(* Logix 5000 project; controller Universal_Device_Info_AOI_V0_1 vendor 1 type 14 code 176 rev 32.11; software revision 32.00; part 2 of 3 *)
(* tags used below, declared in another part *)
   Port : INT;
   Common_Data : Turck_IOLink_Common_Data;
   Universal_IOLink_Info : Universal_IOLink_Info;
   StartupDone : BOOL;
   Done : DINT;
   Error : DINT;
   Active : DINT;
   Pending : DINT;
   Pending_or_Active : DINT;
   MyTicketNum : DINT[32];
   Read_ONS : DINT;
   ReadRequest : DINT;
   Read : DINT;
   DoneCount : DINT;
   Status : DINT;
   ErrorCount : DINT;
   Update_Data : BOOL;
(* Universal_Device_Info, continued *)

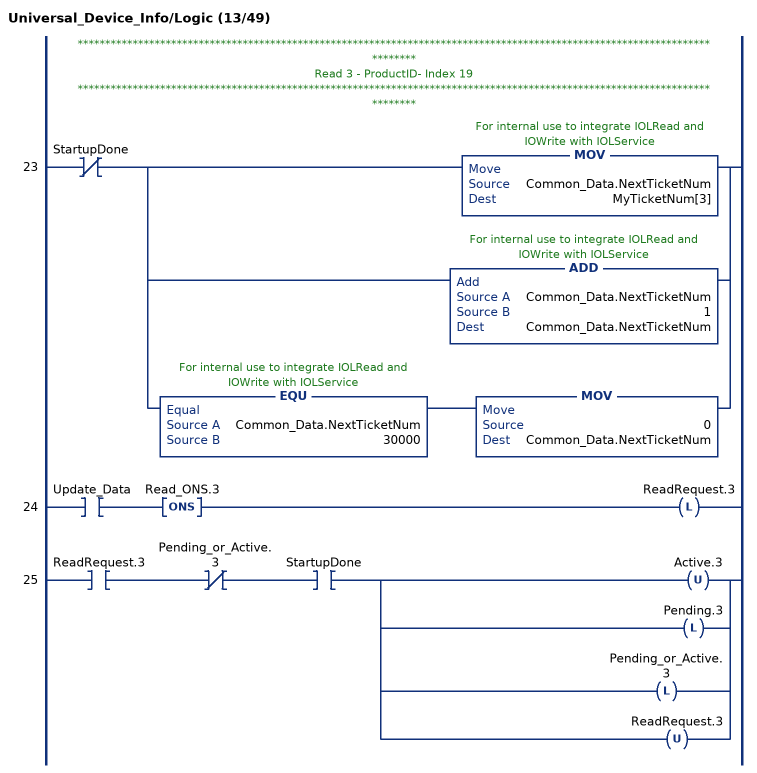
   [picture p25: Universal_Device_Info/Logic rungs 23-25]
   // ***************************************************************************************************************************
   // Read 3 - ProductID- Index 19
   // ***************************************************************************************************************************
   23: XIO(StartupDone)[MOV(Common_Data.NextTicketNum,MyTicketNum[3]) ,ADD(Common_Data.NextTicketNum,1,Common_Data.NextTicketNum) ,EQU(Common_Data.NextTicketNum,30000) MOV(0,Common_Data.NextTicketNum) ];
   24: XIC(Update_Data)ONS(Read_ONS.3)OTL(ReadRequest.3);
   25: XIC(ReadRequest.3)XIO(Pending_or_Active.3)XIC(StartupDone)[OTU(Active.3) ,OTL(Pending.3) ,OTL(Pending_or_Active.3) ,OTU(ReadRequest.3) ];
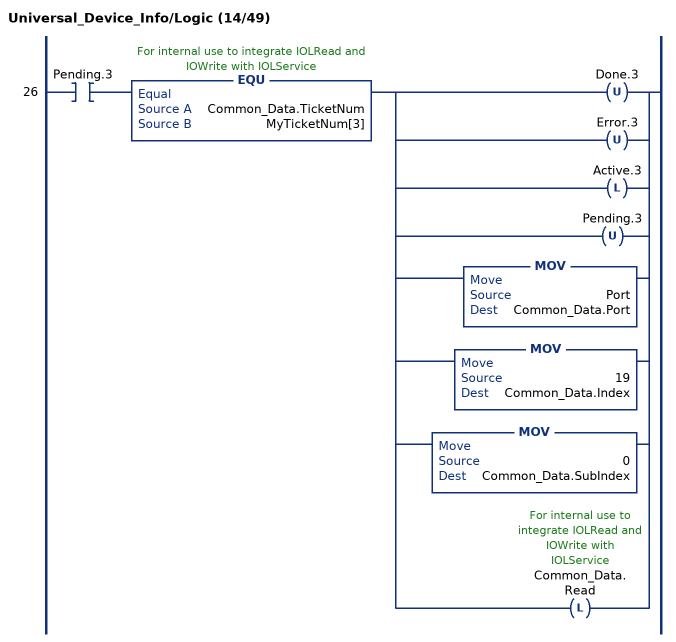
   26: XIC(Pending.3)EQU(Common_Data.TicketNum,MyTicketNum[3])[OTU(Done.3) ,OTU(Error.3) ,OTL(Active.3) ,OTU(Pending.3) ,MOV(Port,Common_Data.Port) ,MOV(19,Common_Data.Index) ,MOV(0,Common_Data.SubIndex) ,OTL(Common_Data.Read) ];
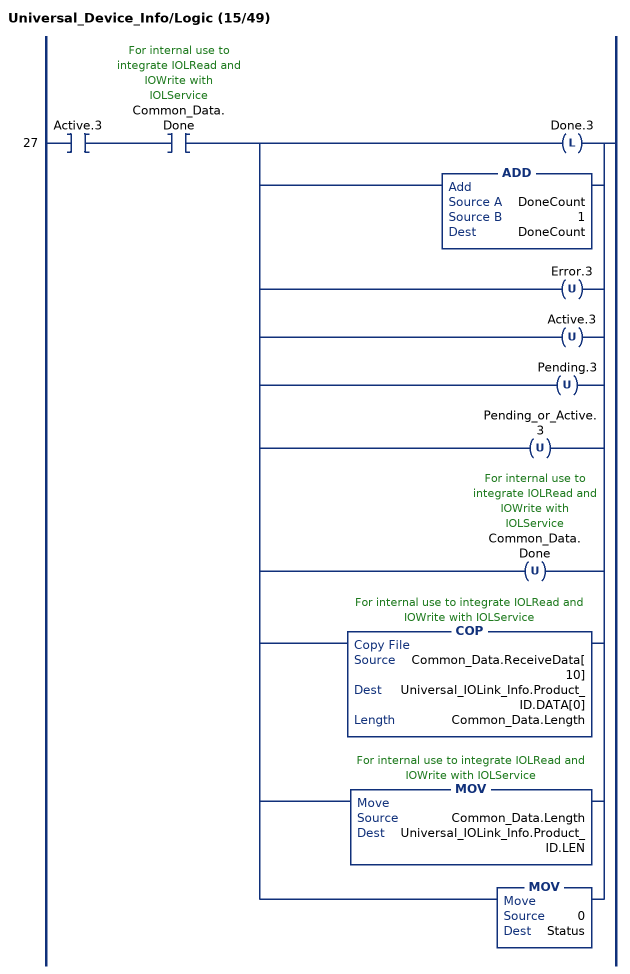
   27: XIC(Active.3)XIC(Common_Data.Done)[OTL(Done.3) ,ADD(DoneCount,1,DoneCount) ,OTU(Error.3) ,OTU(Active.3) ,OTU(Pending.3) ,OTU(Pending_or_Active.3) ,OTU(Common_Data.Done) ,COP(Common_Data.ReceiveData[10],Universal_IOLink_Info.Product_ID.DATA[0],Common_Data.Length) ,MOV(Common_Data.Length,Universal_IOLink_Info.Product_ID.LEN) ,MOV(0,Status) ];
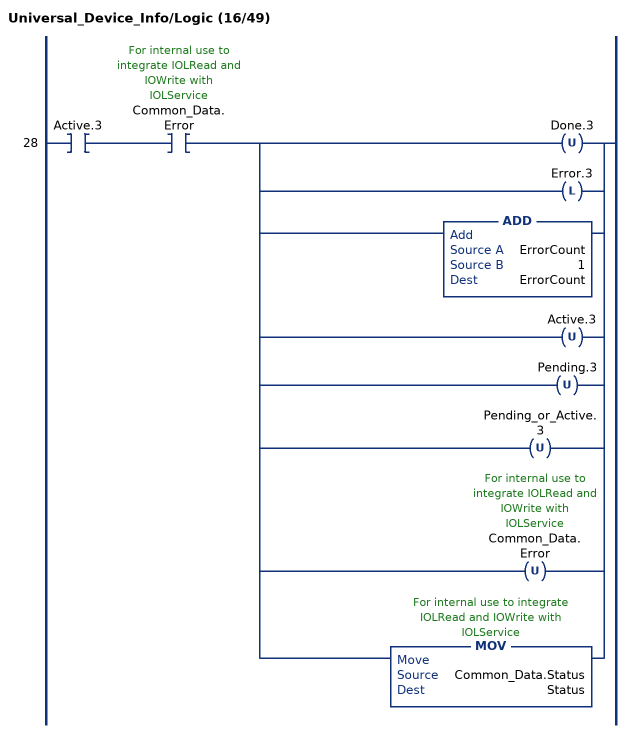
   28: XIC(Active.3)XIC(Common_Data.Error)[OTU(Done.3) ,OTL(Error.3) ,ADD(ErrorCount,1,ErrorCount) ,OTU(Active.3) ,OTU(Pending.3) ,OTU(Pending_or_Active.3) ,OTU(Common_Data.Error) ,MOV(Common_Data.Status,Status) ];
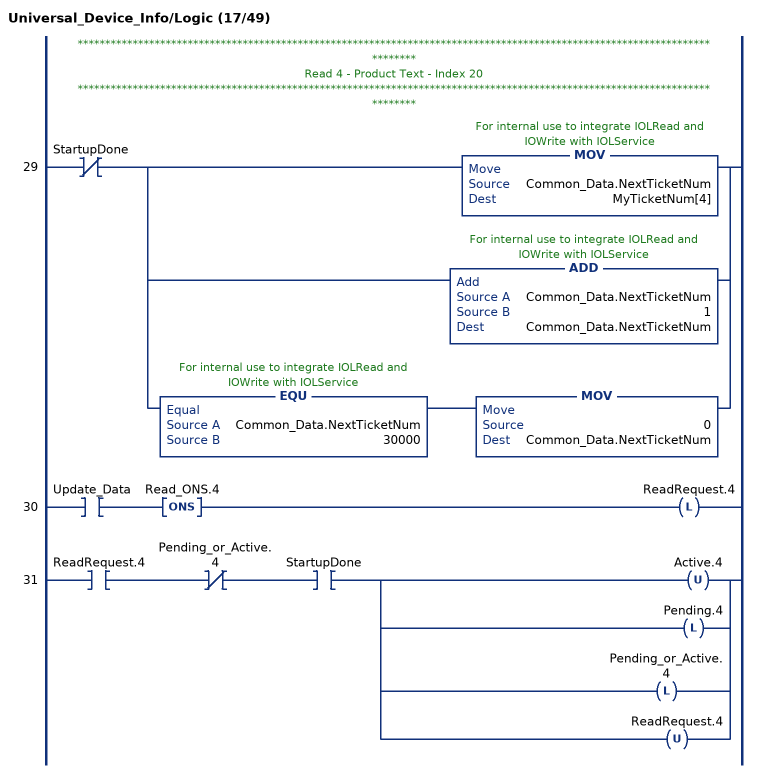
   // ***************************************************************************************************************************
   // Read 4 - Product Text - Index 20
   // ***************************************************************************************************************************
   29: XIO(StartupDone)[MOV(Common_Data.NextTicketNum,MyTicketNum[4]) ,ADD(Common_Data.NextTicketNum,1,Common_Data.NextTicketNum) ,EQU(Common_Data.NextTicketNum,30000) MOV(0,Common_Data.NextTicketNum) ];
   30: XIC(Update_Data)ONS(Read_ONS.4)OTL(ReadRequest.4);
   31: XIC(ReadRequest.4)XIO(Pending_or_Active.4)XIC(StartupDone)[OTU(Active.4) ,OTL(Pending.4) ,OTL(Pending_or_Active.4) ,OTU(ReadRequest.4) ];
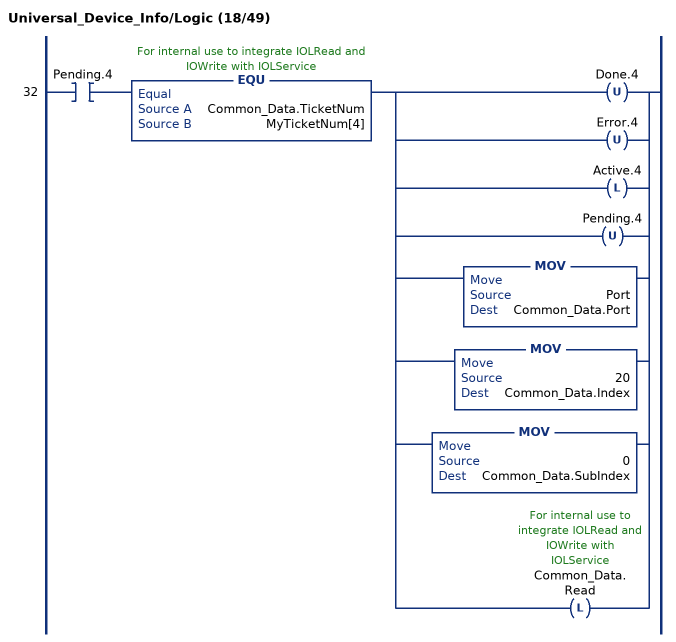
   32: XIC(Pending.4)EQU(Common_Data.TicketNum,MyTicketNum[4])[OTU(Done.4) ,OTU(Error.4) ,OTL(Active.4) ,OTU(Pending.4) ,MOV(Port,Common_Data.Port) ,MOV(20,Common_Data.Index) ,MOV(0,Common_Data.SubIndex) ,OTL(Common_Data.Read) ];
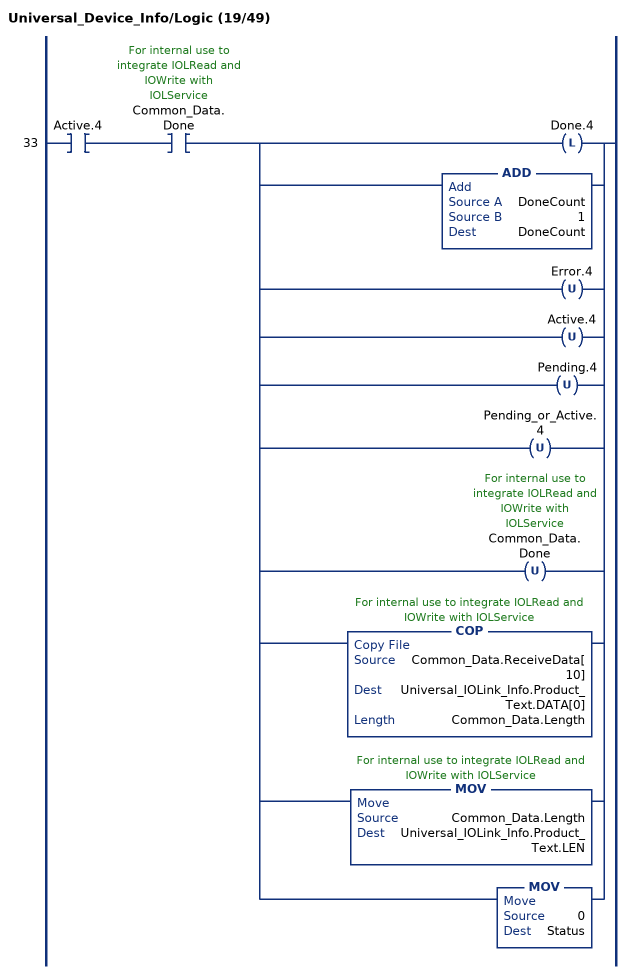
   33: XIC(Active.4)XIC(Common_Data.Done)[OTL(Done.4) ,ADD(DoneCount,1,DoneCount) ,OTU(Error.4) ,OTU(Active.4) ,OTU(Pending.4) ,OTU(Pending_or_Active.4) ,OTU(Common_Data.Done) ,COP(Common_Data.ReceiveData[10],Universal_IOLink_Info.Product_Text.DATA[0],Common_Data.Length) ,MOV(Common_Data.Length,Universal_IOLink_Info.Product_Text.LEN) ,MOV(0,Status) ];
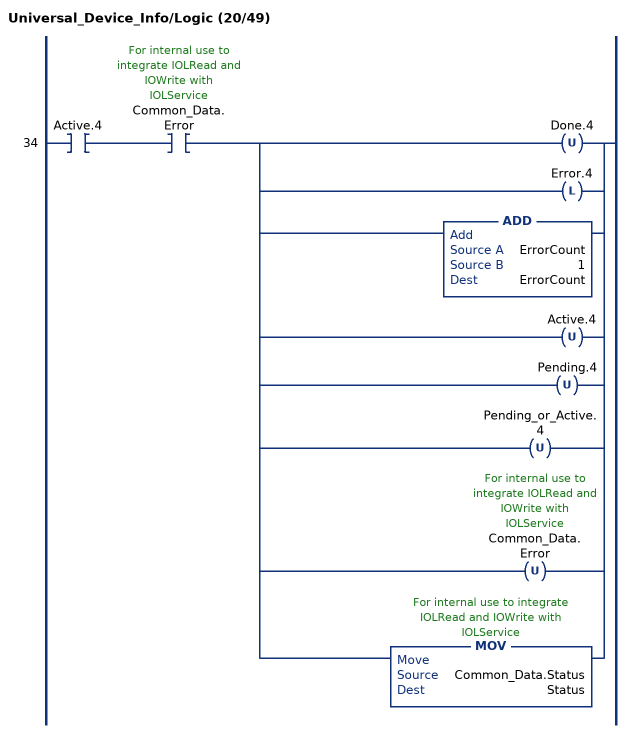
   34: XIC(Active.4)XIC(Common_Data.Error)[OTU(Done.4) ,OTL(Error.4) ,ADD(ErrorCount,1,ErrorCount) ,OTU(Active.4) ,OTU(Pending.4) ,OTU(Pending_or_Active.4) ,OTU(Common_Data.Error) ,MOV(Common_Data.Status,Status) ];
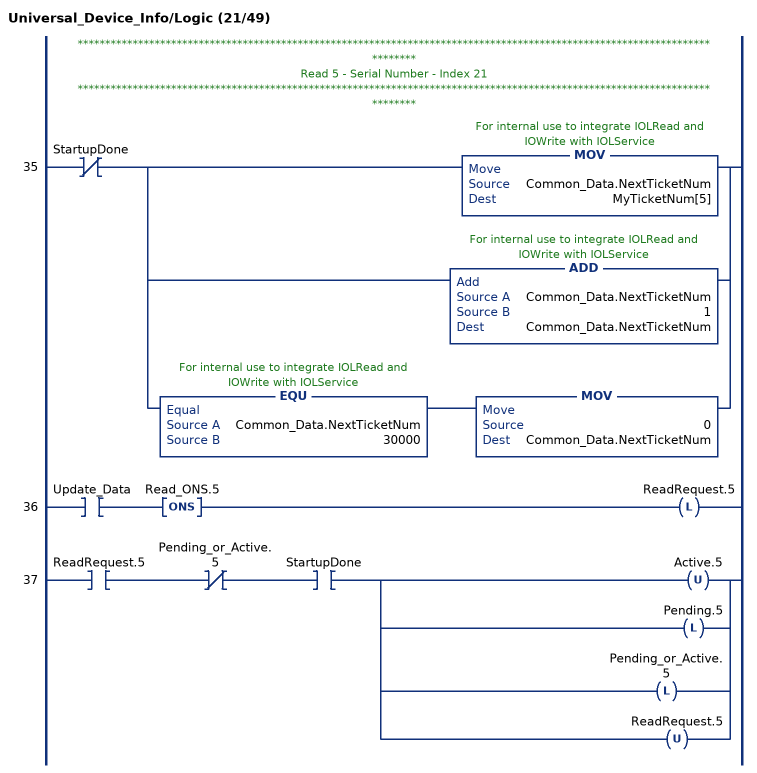
   // ***************************************************************************************************************************
   // Read 5 - Serial Number - Index 21
   // ***************************************************************************************************************************
   35: XIO(StartupDone)[MOV(Common_Data.NextTicketNum,MyTicketNum[5]) ,ADD(Common_Data.NextTicketNum,1,Common_Data.NextTicketNum) ,EQU(Common_Data.NextTicketNum,30000) MOV(0,Common_Data.NextTicketNum) ];
   36: XIC(Update_Data)ONS(Read_ONS.5)OTL(ReadRequest.5);
   37: XIC(ReadRequest.5)XIO(Pending_or_Active.5)XIC(StartupDone)[OTU(Active.5) ,OTL(Pending.5) ,OTL(Pending_or_Active.5) ,OTU(ReadRequest.5) ];
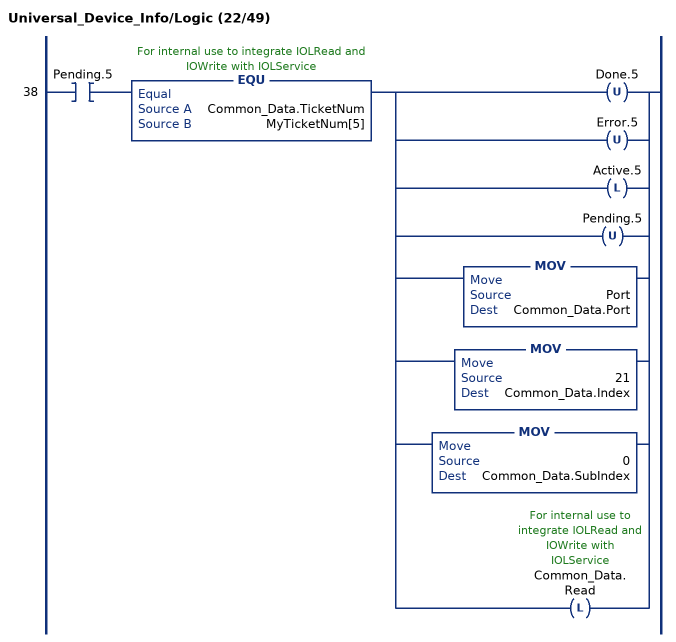
   38: XIC(Pending.5)EQU(Common_Data.TicketNum,MyTicketNum[5])[OTU(Done.5) ,OTU(Error.5) ,OTL(Active.5) ,OTU(Pending.5) ,MOV(Port,Common_Data.Port) ,MOV(21,Common_Data.Index) ,MOV(0,Common_Data.SubIndex) ,OTL(Common_Data.Read) ];
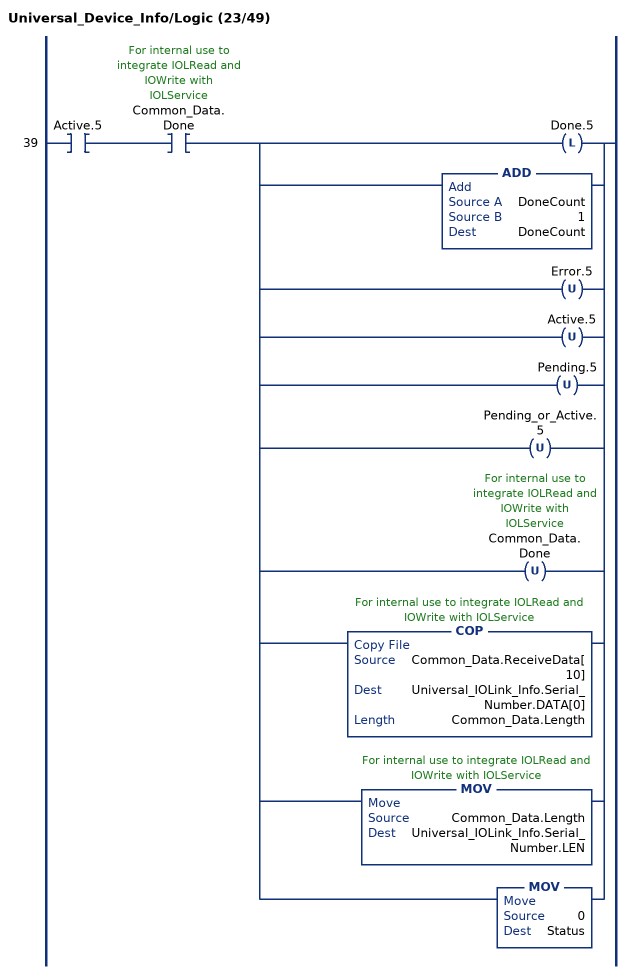
   39: XIC(Active.5)XIC(Common_Data.Done)[OTL(Done.5) ,ADD(DoneCount,1,DoneCount) ,OTU(Error.5) ,OTU(Active.5) ,OTU(Pending.5) ,OTU(Pending_or_Active.5) ,OTU(Common_Data.Done) ,COP(Common_Data.ReceiveData[10],Universal_IOLink_Info.Serial_Number.DATA[0],Common_Data.Length) ,MOV(Common_Data.Length,Universal_IOLink_Info.Serial_Number.LEN) ,MOV(0,Status) ];
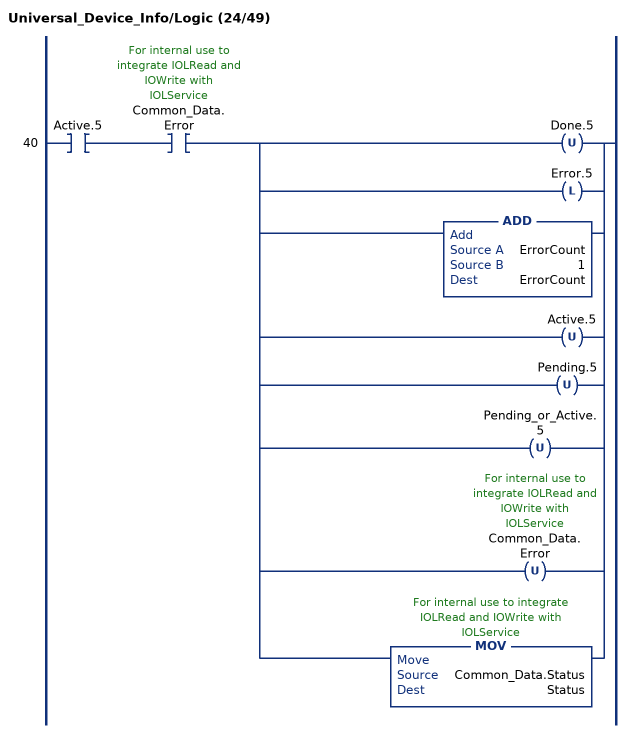
   40: XIC(Active.5)XIC(Common_Data.Error)[OTU(Done.5) ,OTL(Error.5) ,ADD(ErrorCount,1,ErrorCount) ,OTU(Active.5) ,OTU(Pending.5) ,OTU(Pending_or_Active.5) ,OTU(Common_Data.Error) ,MOV(Common_Data.Status,Status) ];
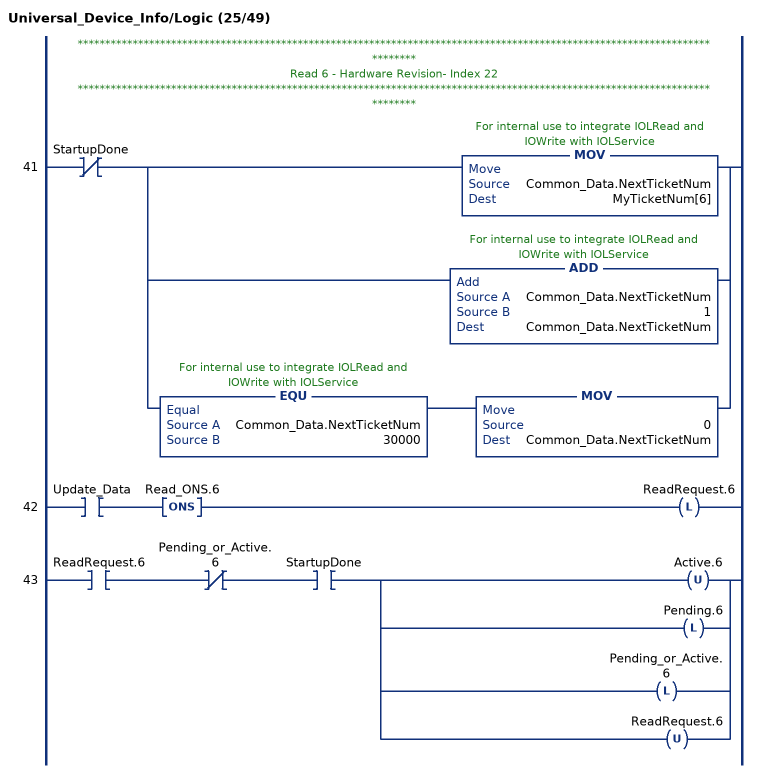
   // ***************************************************************************************************************************
   // Read 6 - Hardware Revision- Index 22
   // ***************************************************************************************************************************
   41: XIO(StartupDone)[MOV(Common_Data.NextTicketNum,MyTicketNum[6]) ,ADD(Common_Data.NextTicketNum,1,Common_Data.NextTicketNum) ,EQU(Common_Data.NextTicketNum,30000) MOV(0,Common_Data.NextTicketNum) ];
   42: XIC(Update_Data)ONS(Read_ONS.6)OTL(ReadRequest.6);
   43: XIC(ReadRequest.6)XIO(Pending_or_Active.6)XIC(StartupDone)[OTU(Active.6) ,OTL(Pending.6) ,OTL(Pending_or_Active.6) ,OTU(ReadRequest.6) ];
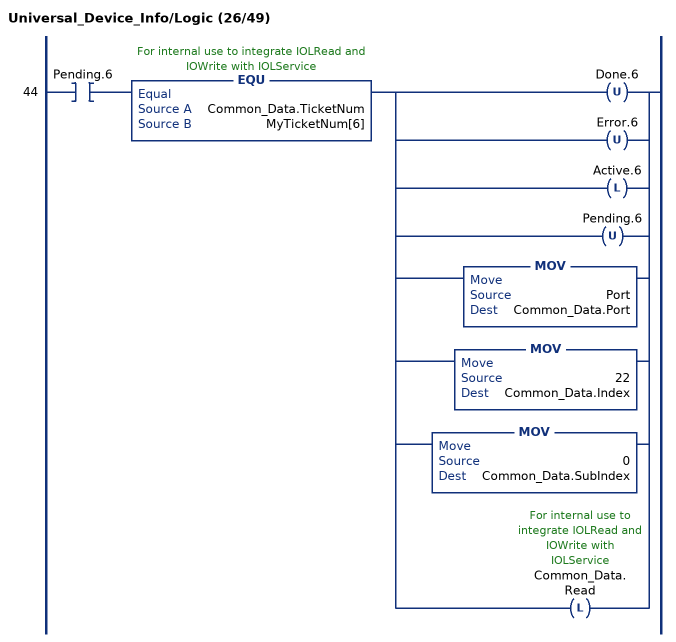
   44: XIC(Pending.6)EQU(Common_Data.TicketNum,MyTicketNum[6])[OTU(Done.6) ,OTU(Error.6) ,OTL(Active.6) ,OTU(Pending.6) ,MOV(Port,Common_Data.Port) ,MOV(22,Common_Data.Index) ,MOV(0,Common_Data.SubIndex) ,OTL(Common_Data.Read) ];
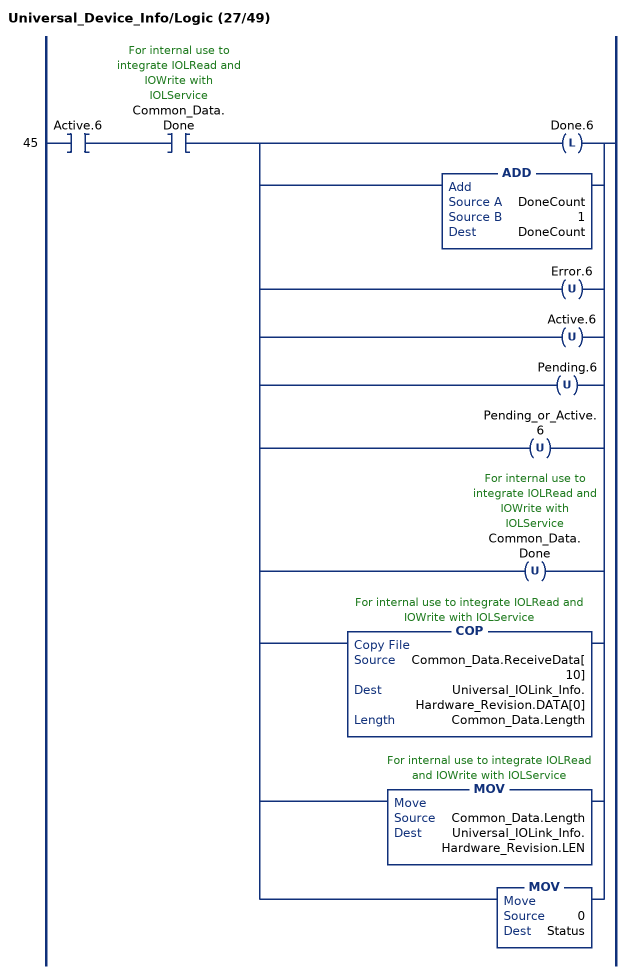
   45: XIC(Active.6)XIC(Common_Data.Done)[OTL(Done.6) ,ADD(DoneCount,1,DoneCount) ,OTU(Error.6) ,OTU(Active.6) ,OTU(Pending.6) ,OTU(Pending_or_Active.6) ,OTU(Common_Data.Done) ,COP(Common_Data.ReceiveData[10],Universal_IOLink_Info.Hardware_Revision.DATA[0],Common_Data.Length) ,MOV(Common_Data.Length,Universal_IOLink_Info.Hardware_Revision.LEN) ,MOV(0,Status) ];
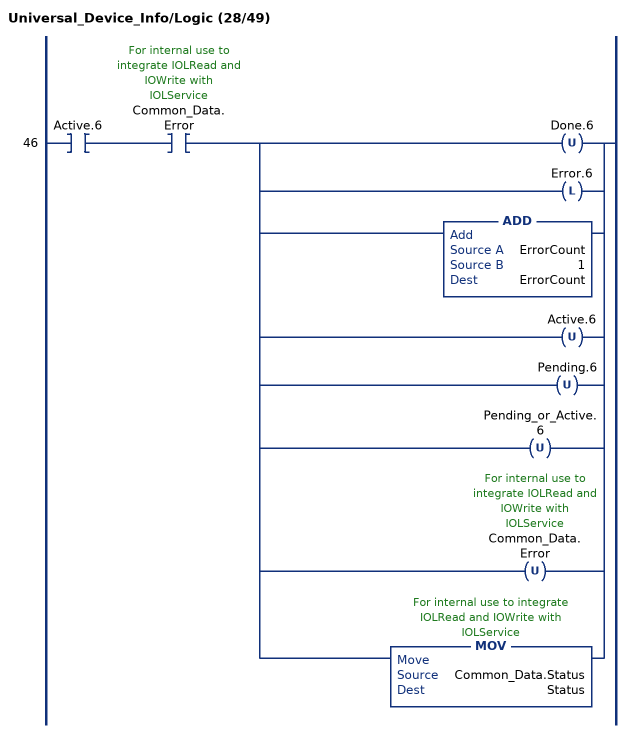
   46: XIC(Active.6)XIC(Common_Data.Error)[OTU(Done.6) ,OTL(Error.6) ,ADD(ErrorCount,1,ErrorCount) ,OTU(Active.6) ,OTU(Pending.6) ,OTU(Pending_or_Active.6) ,OTU(Common_Data.Error) ,MOV(Common_Data.Status,Status) ];
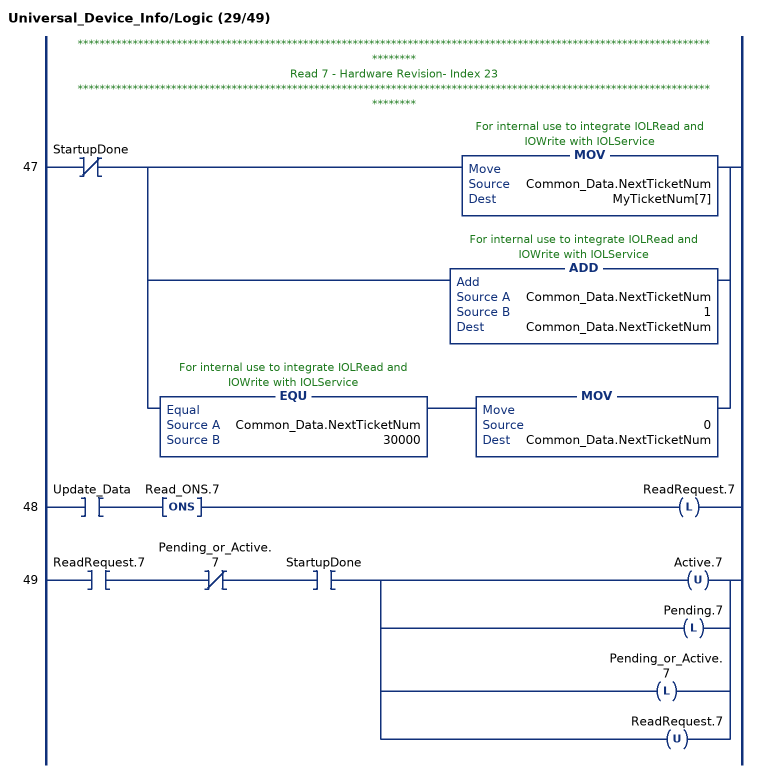
   // ***************************************************************************************************************************
   // Read 7 - Hardware Revision- Index 23
   // ***************************************************************************************************************************
   47: XIO(StartupDone)[MOV(Common_Data.NextTicketNum,MyTicketNum[7]) ,ADD(Common_Data.NextTicketNum,1,Common_Data.NextTicketNum) ,EQU(Common_Data.NextTicketNum,30000) MOV(0,Common_Data.NextTicketNum) ];
   48: XIC(Update_Data)ONS(Read_ONS.7)OTL(ReadRequest.7);
   49: XIC(ReadRequest.7)XIO(Pending_or_Active.7)XIC(StartupDone)[OTU(Active.7) ,OTL(Pending.7) ,OTL(Pending_or_Active.7) ,OTU(ReadRequest.7) ];
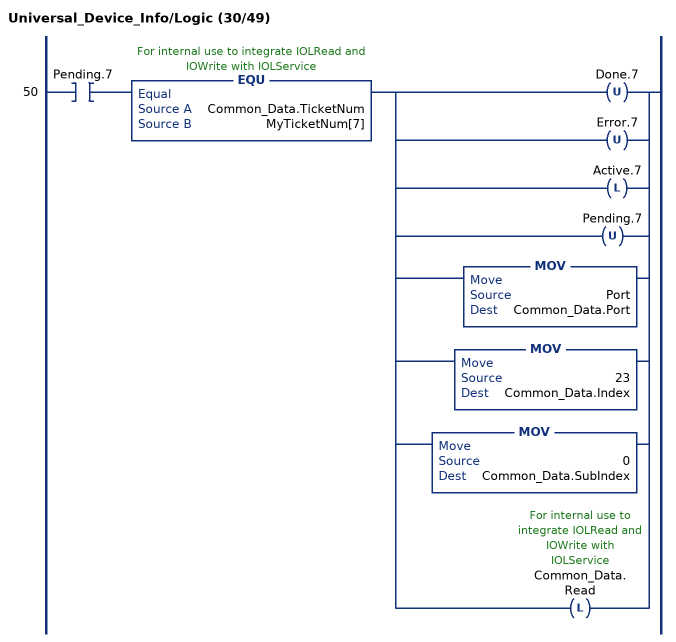
   50: XIC(Pending.7)EQU(Common_Data.TicketNum,MyTicketNum[7])[OTU(Done.7) ,OTU(Error.7) ,OTL(Active.7) ,OTU(Pending.7) ,MOV(Port,Common_Data.Port) ,MOV(23,Common_Data.Index) ,MOV(0,Common_Data.SubIndex) ,OTL(Common_Data.Read) ];
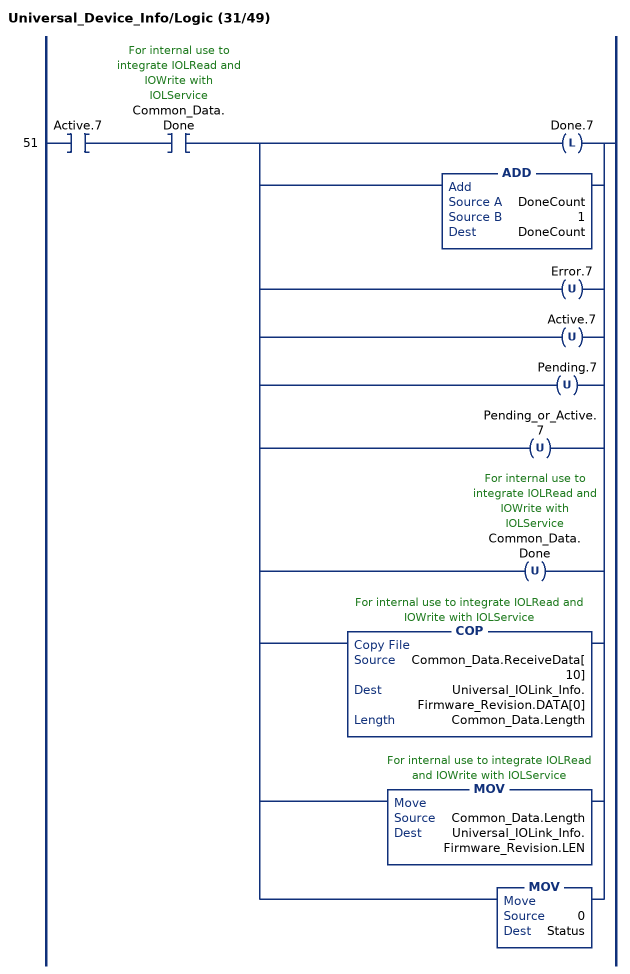
   51: XIC(Active.7)XIC(Common_Data.Done)[OTL(Done.7) ,ADD(DoneCount,1,DoneCount) ,OTU(Error.7) ,OTU(Active.7) ,OTU(Pending.7) ,OTU(Pending_or_Active.7) ,OTU(Common_Data.Done) ,COP(Common_Data.ReceiveData[10],Universal_IOLink_Info.Firmware_Revision.DATA[0],Common_Data.Length) ,MOV(Common_Data.Length,Universal_IOLink_Info.Firmware_Revision.LEN) ,MOV(0,Status) ];
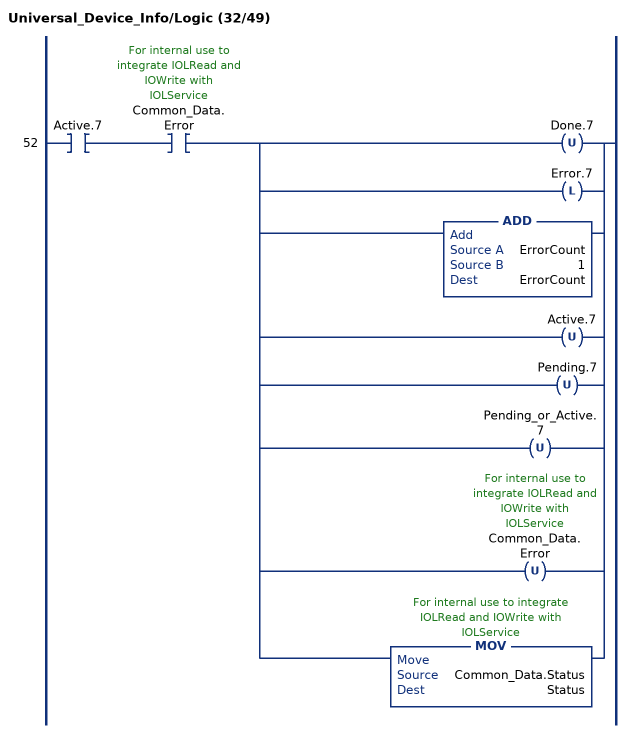
   52: XIC(Active.7)XIC(Common_Data.Error)[OTU(Done.7) ,OTL(Error.7) ,ADD(ErrorCount,1,ErrorCount) ,OTU(Active.7) ,OTU(Pending.7) ,OTU(Pending_or_Active.7) ,OTU(Common_Data.Error) ,MOV(Common_Data.Status,Status) ];
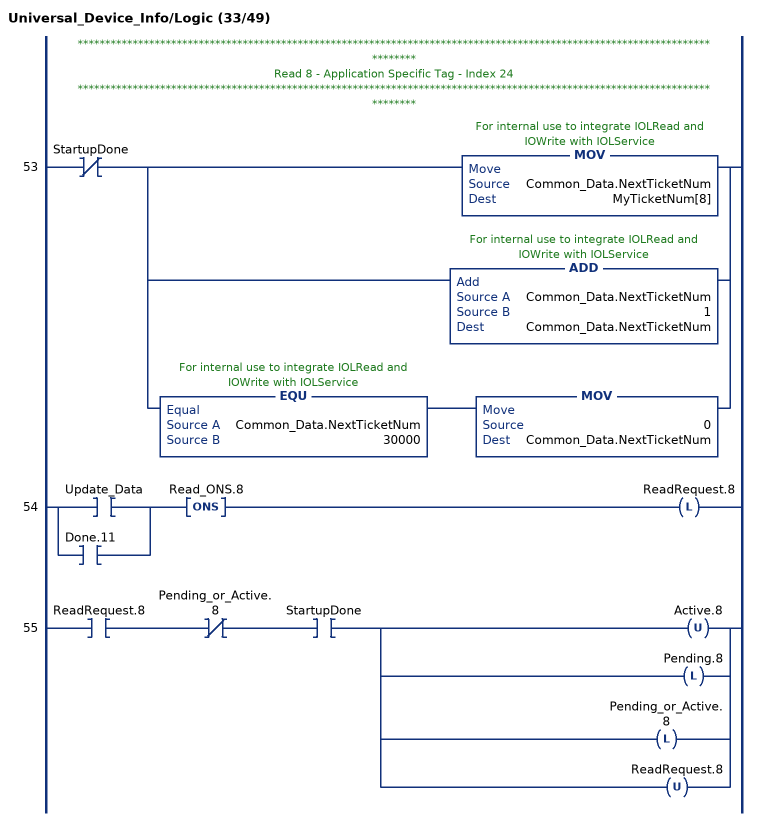
   // ***************************************************************************************************************************
   // Read 8 - Application Specific Tag - Index 24
   // ***************************************************************************************************************************
   53: XIO(StartupDone)[MOV(Common_Data.NextTicketNum,MyTicketNum[8]) ,ADD(Common_Data.NextTicketNum,1,Common_Data.NextTicketNum) ,EQU(Common_Data.NextTicketNum,30000) MOV(0,Common_Data.NextTicketNum) ];
   54: [XIC(Update_Data) ,XIC(Done.11) ]ONS(Read_ONS.8)OTL(ReadRequest.8);
   55: XIC(ReadRequest.8)XIO(Pending_or_Active.8)XIC(StartupDone)[OTU(Active.8) ,OTL(Pending.8) ,OTL(Pending_or_Active.8) ,OTU(ReadRequest.8) ];
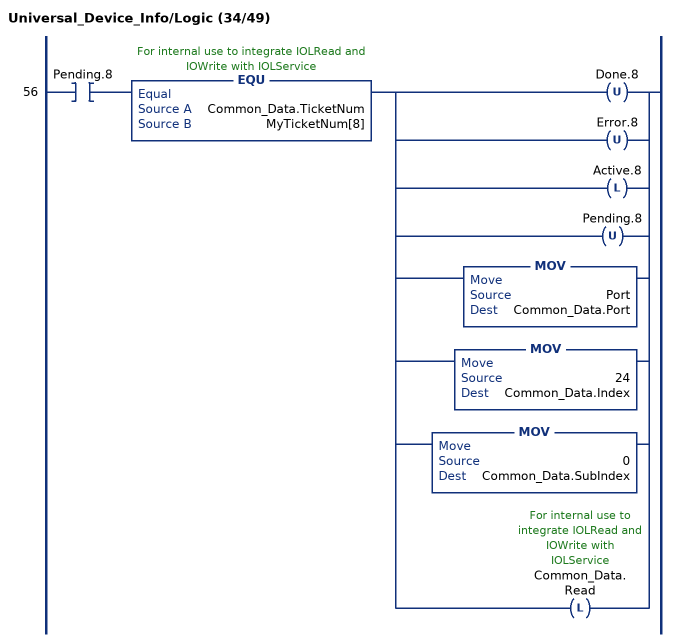
   56: XIC(Pending.8)EQU(Common_Data.TicketNum,MyTicketNum[8])[OTU(Done.8) ,OTU(Error.8) ,OTL(Active.8) ,OTU(Pending.8) ,MOV(Port,Common_Data.Port) ,MOV(24,Common_Data.Index) ,MOV(0,Common_Data.SubIndex) ,OTL(Common_Data.Read) ];
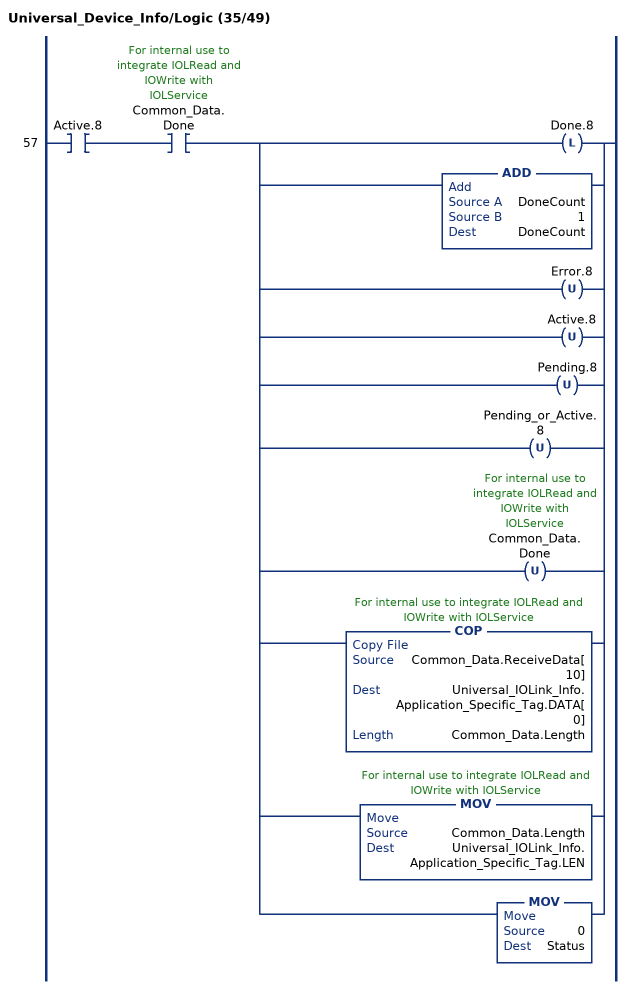
   57: XIC(Active.8)XIC(Common_Data.Done)[OTL(Done.8) ,ADD(DoneCount,1,DoneCount) ,OTU(Error.8) ,OTU(Active.8) ,OTU(Pending.8) ,OTU(Pending_or_Active.8) ,OTU(Common_Data.Done) ,COP(Common_Data.ReceiveData[10],Universal_IOLink_Info.Application_Specific_Tag.DATA[0],Common_Data.Length) ,MOV(Common_Data.Length,Universal_IOLink_Info.Application_Specific_Tag.LEN) ,MOV(0,Status) ];
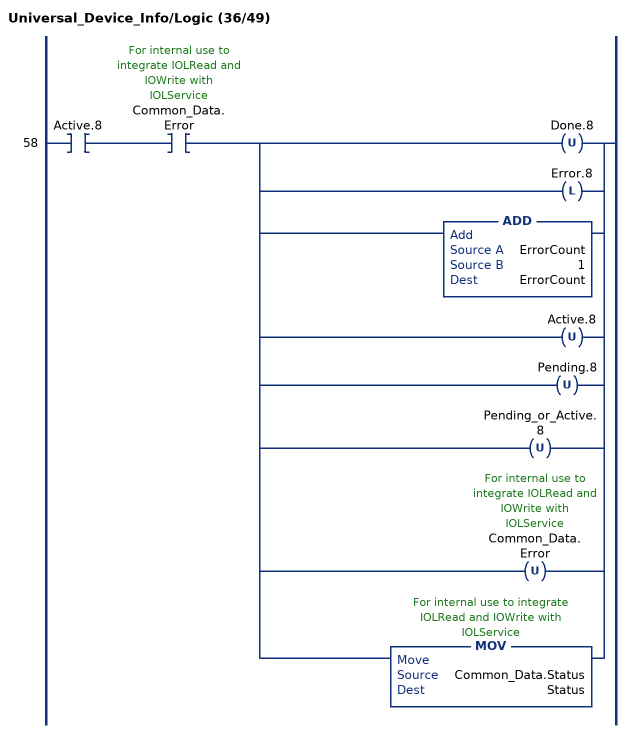
   58: XIC(Active.8)XIC(Common_Data.Error)[OTU(Done.8) ,OTL(Error.8) ,ADD(ErrorCount,1,ErrorCount) ,OTU(Active.8) ,OTU(Pending.8) ,OTU(Pending_or_Active.8) ,OTU(Common_Data.Error) ,MOV(Common_Data.Status,Status) ];
